FUNCTION_BLOCK FB_PayloadPosition
VAR_INPUT
END_VAR
VAR_OUTPUT
END_VAR
VAR
END_VAR

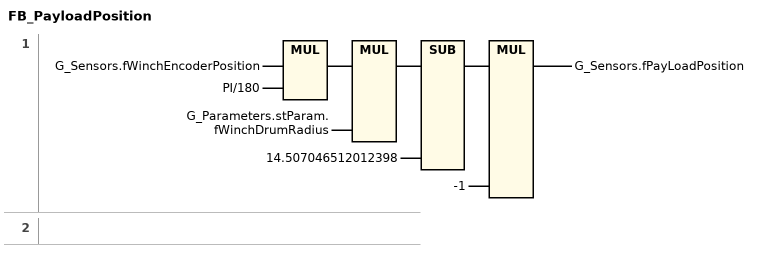
// NETWORK 1
G_Sensors.fPayLoadPosition := ((G_Sensors.fWinchEncoderPosition * (PI/180)) * G_Parameters.stParam.fWinchDrumRadius - 14.507046512012398) * -1;

// NETWORK 2

END_FUNCTION_BLOCK

(* stored: Version 1.1.0.1
   POU FB_PayloadPosition: Id {f696b73c-420f-4ebb-9d47-6ad3abe03394}, SpecialFunc None *)
